(* PLC project cam_2dir_1speed, Dassault Systèmes ControlBuild 2024x *)
(* stored: creationDateTime 2023-10-03T11:13:19-01:00 *)

(* This modules simulates the behaviour of a cam with 2 directions and one speed (ovoid) *)
FUNCTION_BLOCK equipment_library.cam_2dir_1speed
  VAR_INPUT
    forward : BOOL := false;
    backward : BOOL := false;
  END_VAR
  VAR_OUTPUT
    positionTranslat : REAL := 0.0;
    percentTranslat : REAL := 0.0;
    incrementTranslat : REAL := 0.0;
  END_VAR
  VAR_OUTPUT
    angleRotationDeg : REAL := 0.0;
    angleRotationRad : REAL := 0.0;
  END_VAR
  VAR
    firstCycle : BOOL := false;
    incrementRotation : REAL := 0.0;
    memoFwd : BOOL := false;
    memoBwd : BOOL := false;
  END_VAR
  VAR CONSTANT
    maxTranslat : REAL := 1000.0;
    speedVal : REAL := 2.0;
    initTranslat : REAL := 0.0;
    minTranslat : REAL := 0.0;
    oldPosition : REAL := 0.0;
  END_VAR
  VAR
    d_locking : BOOL := false;
    v_d_locking : BOOL := false;
  END_VAR


ACTION C_source_code:
/* ----------------------------------------------------------------	*/
/* Type : Model of Operative Behaviour					*/
/* Category :  Actuators							*/
/* Author : Dassault Systemes						*/
/* Update date : June 2018							*/
/* ----------------------------------------------------------------	*/
/* This module simulate the behaviour of a cam with 2 directions and	*/
/* 1 speed.									*/
/* The position of the cam goes from minTranslat to maxTranslat with	*/
/* the rotation speed speedVal.						*/
/*										*/
/* nota : the starting position is forced by initTranslat.		*/
/* ----------------------------------------------------------------	*/

/* Declaration of variables which don't need to be visualized during simulation */
float pi=3.1415926;



/* ----------------------------------------------------------------	*/
/* Initialization of the position of the cam for the first step of	*/
/* simulation.								*/
/* ----------------------------------------------------------------	*/
if (! firstCycle) {
	if (initTranslat > maxTranslat) positionTranslat = maxTranslat;
	else
		if (initTranslat < minTranslat) positionTranslat = minTranslat;
		else positionTranslat = initTranslat;

	firstCycle = 1;
	if ((maxTranslat - minTranslat) != 0.0)
		angleRotationRad = acos(1 - ((positionTranslat - minTranslat)/(maxTranslat - minTranslat)*2.0));
}

/* ----------------------------------------------------------------	*/
/* Manage priorities of inputs' switching					*/
/* ----------------------------------------------------------------	*/
if (forward && !memoBwd) memoFwd = 1;
if (!forward) memoFwd = 0;
if (!memoFwd && backward) memoBwd= 1;
if (!backward) memoBwd = 0;


/* ----------------------------------------------------------------	*/
/* Rotation and translation (height of cam)				*/
/* ----------------------------------------------------------------	*/
if ((!d_locking) && (memoFwd || memoBwd)) {

	/* compute the increment of rotation according to the clock of simulation	*/
	incrementRotation= speedVal * (CLOCK_PERIOD/1000000);

	/* compute the angle of rotation (radian)	*/
	if (memoFwd) angleRotationRad = angleRotationRad + incrementRotation;
	if (memoBwd) angleRotationRad = angleRotationRad - incrementRotation;
	if (angleRotationRad >= (2*pi)) {angleRotationRad -= 2*pi;}
	
	/* compute the position of translation	*/
	positionTranslat=(1 - cos(angleRotationRad))*(maxTranslat-minTranslat)/2.0 + minTranslat;
}

/* ----------------------------------------------------------------	*/
/* Compute the pecentage of height between the current position	*/
/* and the lowest and highest points of the cam				*/
/* ----------------------------------------------------------------	*/
percentTranslat = (100/(maxTranslat - minTranslat)) * (positionTranslat - minTranslat)  ;
		
/* ----------------------------------------------------------------	*/
/* Conversion of the rotation angle from radian to degree		*/
/* ----------------------------------------------------------------	*/
angleRotationDeg = (angleRotationRad*180)/pi;

/* ----------------------------------------------------------------	*/
/* Increment of translation							*/
/* ----------------------------------------------------------------	*/
incrementTranslat = positionTranslat - oldPosition;
oldPosition = positionTranslat;
END_ACTION

ACTION C_header:
#include <math.h>
END_ACTION
END_FUNCTION_BLOCK
